// TIA Portal V20 export
TYPE "LKinCtrl_TypePnPDiagnostics"
   STRUCT
      status : Word;   // Block status
      subFunctionStatus : Word;   // Status of the subfunction
      stateNumber : DInt;   // State number
      additionalValue1 : Word;   // Additional status information
      additionalValue2 : Word;   // Additional status information
   END_STRUCT;
END_TYPE
